FUNCTION_BLOCK PAEAmmeter EXTENDS PAESensorAnalog
VAR_INPUT
END_VAR
VAR_OUTPUT
END_VAR
VAR
END_VAR

END_FUNCTION_BLOCK

(* stored: Version 1.1.0.1, ProductVersion 3.1.4020.6
   POU PAEAmmeter: Id {598b7c52-afb0-4fac-b07a-6ba782c43600}, SpecialFunc None *)
